// TwinCAT 3 PLC project PLC1
// ProgramVersion: 3.1.4023.0
// libraries:
//   Tc2_ModbusRTU, * (Beckhoff Automation GmbH)
//   Tc2_Standard, * (Beckhoff Automation GmbH)
//   Tc2_System, * (Beckhoff Automation GmbH)
//   Tc2_Utilities, * (Beckhoff Automation GmbH)
//   Tc3_Module, * (Beckhoff Automation GmbH)
// project tree:
//   / PlcTask.TcTTO
//   POUs/ FB_ModbusMaster.TcPOU, FB_ModbusSlave.TcPOU, FB_PM2200.TcPOU, FB_TDS3000.TcPOU, I_ModbusSlave.TcIO, MAIN.TcPOU
// real-time tasks:
//   TASK PlcTask: cycle T#50us, priority 20, ADS port 350
// I/O:
//   DEVICE Device 1 (COM Port)
//   DEVICE Device 2 (EtherCAT), AmsNetId 192.168.56.1.3.1
//     Term 1 (EK1100) [EK1100 EtherCAT Coupler (2A E-Bus)]
//       Term 2 (EL6022) [EL6022 Interface 2Ch. (RS422/485)]
// variable links:
//   PLC1/PLC1 Instance <-> Device 1 (COM Port)
//     PlcTask Inputs/MAIN.fbModbusMaster.fbModbusMaster.InData/D <-> Inputs/Data1
//     PlcTask Inputs/MAIN.fbModbusMaster.fbModbusMaster.InData/D @bit {8..504 step 8} <-> Inputs/Data{2..64}  (63 links)
//     PlcTask Inputs/MAIN.fbModbusMaster.fbModbusMaster.InData/SerStatus <-> Inputs/Status
//     PlcTask Outputs/MAIN.fbModbusMaster.fbModbusMaster.OutData/D <-> Outputs/Data1
//     PlcTask Outputs/MAIN.fbModbusMaster.fbModbusMaster.OutData/D @bit {8..504 step 8} <-> Outputs/Data{2..64}  (63 links)
//     PlcTask Outputs/MAIN.fbModbusMaster.fbModbusMaster.OutData/SerCtrl <-> Outputs/Ctrl

CONFIGURATION PLC1
    RESOURCE PLC ON TwinCAT3
        TASK PlcTask(INTERVAL := T#50us, PRIORITY := 20);
        PROGRAM MAIN WITH PlcTask : MAIN;
    END_RESOURCE
END_CONFIGURATION

// ---- POUs/I_ModbusSlave.TcIO
INTERFACE I_ModbusSlave

PROPERTY Address : POINTER TO WORD
GET
END_GET
END_PROPERTY

METHOD Convert : BOOL
VAR_INPUT
	iRegionNo	:	INT;
	pReadData	:	POINTER TO BYTE;
END_VAR
END_METHOD

METHOD FirstCycle : BOOL
VAR_INPUT
END_VAR
END_METHOD

PROPERTY Name : STRING
GET
END_GET
SET
END_SET
END_PROPERTY

PROPERTY NumAddRegion : UINT
GET
END_GET
END_PROPERTY

PROPERTY UnitID : BYTE
GET
END_GET
SET
END_SET
END_PROPERTY

END_INTERFACE

// ---- POUs/MAIN.TcPOU
PROGRAM MAIN
VAR
	fbModbusMaster 	:		FB_ModbusMaster;
	fbModbusSlave	:		FB_PM2200;
	fbModbusTemp	: 		FB_TDS3000;
	istep			:		UINT;
	bStart			:		BOOL;
	
	arrData			:		ARRAY [0..255] OF BYTE;
END_VAR

CASE istep OF
	0: //Trigger
		IF bStart THEN
			bStart := FALSE;
			istep := 10;
		END_IF
		
	10: //Init
		fbModbusSlave.UnitID := 1;
		fbModbusSlave.FirstCycle();
		fbModbusTemp.UnitID := 2;
		fbModbusTemp.FirstCycle();
		
		fbModbusMaster.FirstCycle();
		fbModbusMaster.Init();
		fbModbusMaster.RegisterSlave(fbModbusSlave);
		fbModbusMaster.RegisterSlave(fbModbusTemp);
		fbModbusMaster.Timeout := 1000;
		istep := 20;
		
	20: //Running
		IF fbModbusMaster.Run() THEN
			istep := 30;
		END_IF
		
	30: //Stopped
		
END_CASE

fbModbusMaster();

END_PROGRAM

// ---- POUs/FB_ModbusMaster.TcPOU
FUNCTION_BLOCK FB_ModbusMaster //IMPLEMENTS I_UniversalUnit
VAR
	sName			:		STRING;
	bInitialized	:		BOOL;
	iScantime		:		UINT;
	iTimeout		:		UINT;
	iErrorID		:		UDINT;
	
	bBusy			: 		BOOL;
	bError			:		BOOL;
	
	iStepInit		:		INT;
	iStepGeneral	: 		INT;
	iStepRunning	:		INT;
	bFirstCycle		:		BOOL;
	
	bRun			:		BOOL;
	bStop			: 		BOOL;
	
	fbModbusMaster	: 		ModbusRtuMaster_PcCOM;
	ipModbusSlave	:		ARRAY [1..247] OF I_ModbusSlave;
	iAmountSlave	: 		UINT;
	
	iLoopSlave		:		UINT	:= 1;
	iLoopAdr		:		UINT;
	iQuantity 		: 		POINTER TO WORD;
	iMBAddr 		: 		POINTER TO WORD;
    arrData			: 		ARRAY [0..255] OF BYTE;
	
END_VAR

IF bFirstCycle THEN
	bFirstCycle := FALSE;
END_IF
		
StateMachine();

bRun := FALSE;
bStop := FALSE;

bInitialized := iStepGeneral >= 20;

bError := fbModbusMaster.Error AND iStepGeneral = 30;
iErrorID := fbModbusMaster.ErrorId;
bBusy := fbModbusMaster.BUSY AND iStepGeneral = 30;

//	// error	
//		fbAxisError.Description := FUN_MergeStrings5(sMotorName, ' axis error number: ', UDINT_TO_STRING(iErrorID), '', '');
//		fbAxisError.Set(bError);

METHOD Abort : BOOL
END_METHOD

PROPERTY AnyError : BOOL
GET
AnyError 	:= bError;
END_GET
END_PROPERTY

PROPERTY Busy : BOOL
GET
Busy := bBusy;
END_GET
END_PROPERTY

PROPERTY ErrorID : UDINT
GET
ErrorID := iErrorID;
END_GET
END_PROPERTY

METHOD FirstCycle : BOOL
VAR_INPUT
//	ipAlarmController	: I_AlarmController;
//	ipHMIController	: I_HMIController;
END_VAR
END_METHOD

METHOD Init : BOOL
IF iStepGeneral = 0 THEN
	iStepGeneral := 10;
END_IF

//Method output
	Init := (iStepGeneral >= 20);
END_METHOD

PROPERTY Initialized : BOOL
GET
Initialized := bInitialized;
END_GET
END_PROPERTY

PROPERTY Name : STRING
GET
Name := sName;
END_GET
SET
sName := Name;
END_SET
END_PROPERTY

PROPERTY ReadData : ARRAY [0..255] OF BYTE
GET
ReadData := arrData;
END_GET
END_PROPERTY

PROPERTY ReadDataSize : uint
GET
ReadDataSize := INT_TO_UINT(SIZEOF(arrData));
END_GET
END_PROPERTY

METHOD RegisterSlave : BOOL
VAR_INPUT
	ModbusSlave		:		I_ModbusSlave;
END_VAR
VAR
	iLoop	:	UINT;
	bExists	:	BOOL;
END_VAR
FOR iLoop := 1 TO iAmountSlave DO
	IF ipModbusSlave[iLoop] = ModbusSlave THEN
		bExists := TRUE;
		iLoop := iAmountSlave;
	END_IF
END_FOR 
IF NOT bExists THEN
	iAmountSlave := iAmountSlave + 1;
	ipModbusSlave[iAmountSlave] := ModbusSlave;
END_IF
END_METHOD

METHOD Reset : BOOL
bError := FALSE;
iErrorID := 0;
bError := FALSE;
iStepInit		:= 0;
iStepGeneral	:= 0;
iStepRunning	:= 0;

iLoopSlave		:= 1;
iLoopAdr		:= 0;

fbModbusMaster.Execute := FALSE;

Reset := TRUE;
END_METHOD

METHOD Run : BOOL
IF (iStepGeneral = 20) THEN
	iStepGeneral := 30;
END_IF

bRun := TRUE;
Run := (iStepGeneral >= 30) AND (iStepGeneral < 200);
END_METHOD

PROPERTY ScanTime : UINT
GET
ScanTime := iScantime;
END_GET
SET
iScantime := ScanTime;
END_SET
END_PROPERTY

METHOD StateInit : BOOL (*Unit is performing initialization*)
IF NOT bError THEN
	iStepGeneral := 20;
END_IF
END_METHOD

METHOD StateMachine : BOOL (*State machine of unit*)
//State machine						   
	CASE iStepGeneral OF
		0:  //Uninitialized
			StateUninitialized();
	
		10: //Initializing
			StateInit();
	
		20: //Ready
			StateReady();
		
		30: //Running
			StateRunning();
						
		200: //stop
			StateStopping();
			
		210: //stop done
			StateStoppingDone();
	END_CASE
END_METHOD

METHOD StateReady : BOOL (* Unit is initialized*)
END_METHOD

METHOD StateRunning : BOOL (* Unit is uninitialized*)
VAR 
END_VAR
CASE iStepRunning OF
	0: // Trigger
		IF iAmountSlave > 0 THEN
			iStepRunning := 10;
		ELSE
			iStepRunning := 50;
		END_IF
		
	10: // Set parameters
		IF iLoopSlave <= iAmountSlave THEN
			IF  iLoopAdr <= ipModbusSlave[iLoopSlave].NumAddRegion - 1 THEN
				iQuantity := (ipModbusSlave[iLoopSlave].Address + (iLoopAdr*2+1)*SIZEOF(WORD));
				iMBAddr := (ipModbusSlave[iLoopSlave].Address + (iLoopAdr*2)*SIZEOF(WORD));
				
				fbModbusMaster.UnitID 	:=		ipModbusSlave[iLoopSlave].UnitID;
				fbModbusMaster.Quantity	:=		iQuantity^;
				fbModbusMaster.MBAddr	:=		iMBAddr^;
				fbModbusMaster.cbLength	:= 		SIZEOF(arrData);
				fbModbusMaster.pMemoryAddr	:= 	ADR(arrData);
				fbModbusMaster.Timeout	:= 		UINT_TO_TIME(iTimeout);
				
				iLoopAdr := iLoopAdr + 1;
			ELSE
				iLoopAdr := 0;
				iLoopSlave := iLoopSlave + 1;
			END_IF
		ELSE
			iLoopSlave := 1;
		END_IF
		iStepRunning := 20;
		
	20: // Send request
		IF NOT fbModbusMaster.BUSY THEN
			iStepRunning := 30;
		END_IF
	
	30: // Wait ack request
		IF fbModbusMaster.BUSY THEN
			iStepRunning := 40;
		END_IF
		
	40: // Wait respond
		IF NOT fbModbusMaster.BUSY THEN
			iStepRunning := 50;
		END_IF
		
	50: // Convert raw data
		ipModbusSlave[iLoopSlave].Convert(iLoopAdr, ADR(arrData));

	60: // Return, done
		iStepRunning := 0;
		
END_CASE

IF (iStepRunning >= 20) AND (iStepRunning <= 40) THEN
	fbModbusMaster.ReadRegs();
END_IF
fbModbusMaster.Execute := iStepRunning >= 20 AND iStepRunning <= 30;


//bTest S= iStepRunning > 
//tonTest(IN :=
END_METHOD

METHOD StateStopping : BOOL (* Unit is uninitialized*)
iStepGeneral	:= 0;
iStepRunning	:= 210;

iLoopSlave		:= 1;
iLoopAdr		:= 0;

fbModbusMaster.Execute := FALSE;
END_METHOD

METHOD StateStoppingDone : BOOL (* Unit is uninitialized*)
IF NOT bStop THEN
	iStepGeneral := 20;
END_IF
END_METHOD

METHOD StateUninitialized : BOOL (* Unit is uninitialized*)
END_METHOD

METHOD Stop : BOOL
IF iStepGeneral >= 30 AND iStepGeneral < 200 THEN
	iStepGeneral := 200;
END_IF
bStop := TRUE;

Stop := (iStepGeneral = 210);
END_METHOD

PROPERTY Timeout : UINT
GET
Timeout := iTimeout;
END_GET
SET
iTimeout := Timeout;
END_SET
END_PROPERTY

END_FUNCTION_BLOCK

// ---- POUs/FB_PM2200.TcPOU
FUNCTION_BLOCK FB_PM2200 EXTENDS FB_ModbusSlave
VAR
	arrAccPower	:	ARRAY [0..41] OF WORD;
	arrQuaPower		:	ARRAY [0..17] OF WORD;
	arrCommon		:	ARRAY [0..111] OF WORD;
END_VAR

PROPERTY AccPower : ARRAY [0..41] OF WORD
GET
AccPower := arrAccPower;
END_GET
END_PROPERTY

PROPERTY Common : ARRAY [0..111] OF WORD
GET
Common := arrCommon;
END_GET
END_PROPERTY

METHOD Convert : BOOL
VAR_INPUT
	iRegionNo	:	INT;
	pReadData	:	POINTER TO BYTE;
END_VAR
VAR
	pTempData	: 	POINTER TO BYTE;
	iTempData	: 	BYTE;
	iLoop		: 	INT;
	bHiByte		:	BOOL := TRUE;
END_VAR
CASE iRegionNo OF
	0: 
		FOR iLoop := 0 TO SIZEOF(arrAccPower)*2 DO
			pTempData := (pReadData + iLoop);
			iTempData := pTempData^;
			
			IF bHiByte THEN
				arrAccPower[iLoop/2] := SHL(BYTE_TO_WORD(iTempData), 8);
			ELSE 
				arrAccPower[iLoop/2] := arrAccPower[iLoop/2] + BYTE_TO_WORD(iTempData);
				IF bSwap THEN
					arrAccPower[iLoop/2] := ROL(arrAccPower[iLoop/2], 8);
				END_IF
			END_IF
			bHiByte := NOT bHiByte;
		END_FOR
		
	1: 
		FOR iLoop := 0 TO SIZEOF(arrQuaPower)*2 DO
			pTempData := (pReadData + iLoop);
			iTempData := pTempData^;
			
			IF bHiByte THEN
				arrQuaPower[iLoop/2] := SHL(BYTE_TO_WORD(iTempData), 8);
			ELSE 
				arrQuaPower[iLoop/2] := arrQuaPower[iLoop/2] + BYTE_TO_WORD(iTempData);
				IF bSwap THEN
					arrQuaPower[iLoop/2] := ROL(arrQuaPower[iLoop/2], 8);
				END_IF
			END_IF
			bHiByte := NOT bHiByte;
		END_FOR

	2: 
		FOR iLoop := 0 TO SIZEOF(arrCommon)*2 DO
			pTempData := (pReadData + iLoop);
			iTempData := pTempData^;
			
			IF bHiByte THEN
				arrCommon[iLoop/2] := SHL(BYTE_TO_WORD(iTempData), 8);
			ELSE 
				arrCommon[iLoop/2] := arrCommon[iLoop/2] + BYTE_TO_WORD(iTempData);
				IF bSwap THEN
					arrCommon[iLoop/2] := ROL(arrCommon[iLoop/2], 8);
				END_IF
			END_IF
			bHiByte := NOT bHiByte;
		END_FOR

END_CASE
END_METHOD

METHOD FirstCycle : BOOL
VAR_INPUT
END_VAR
arrAddress[0][0] := 2999;			// Current
arrAddress[0][1] := 12;

arrAddress[1][0] := 3019;			// Voltage
arrAddress[1][1] := 14;		
		
arrAddress[2][0] := 3053;
arrAddress[2][1] := 16;				// Power
arrAddress[3][0] := 3069;
arrAddress[3][1] := 8;				

arrAddress[4][0] := 3077;			// Power factor
arrAddress[4][1] := 16;		
		
arrAddress[5][0] := 3109;			// Frequency
arrAddress[6][1] := 2;				

iNumAddRegion := 6;
END_METHOD

PROPERTY QuaPower : ARRAY [0..17] OF WORD
GET
QuaPower := arrQuaPower;
END_GET
END_PROPERTY

END_FUNCTION_BLOCK

// ---- POUs/FB_ModbusSlave.TcPOU
FUNCTION_BLOCK FB_ModbusSlave IMPLEMENTS I_ModbusSlave
VAR
	iUnitID			: 		BYTE;
	arrAddress		:		ARRAY [0..20] OF ARRAY [0..1] OF WORD;
	iNumAddRegion	:		UINT;
	bSwap			:		BOOL;
	
	sName			:		STRING;

END_VAR

PROPERTY Address : POINTER TO WORD
GET
Address := ADR(arrAddress);
END_GET
END_PROPERTY

METHOD Convert : BOOL
VAR_INPUT
	iRegionNo	:	INT;
	pReadData	:	POINTER TO BYTE;
END_VAR
END_METHOD

METHOD FirstCycle : BOOL
VAR_INPUT
END_VAR
END_METHOD

PROPERTY Name : STRING
GET
Name := sName;
END_GET
SET
sName := Name;
END_SET
END_PROPERTY

PROPERTY NumAddRegion : UINT
GET
NumAddRegion := iNumAddRegion;
END_GET
END_PROPERTY

PROPERTY UnitID : BYTE
GET
UnitID := iUnitID;
END_GET
SET
iUnitID := UnitID;
END_SET
END_PROPERTY

END_FUNCTION_BLOCK

// ---- POUs/FB_TDS3000.TcPOU
FUNCTION_BLOCK FB_TDS3000 EXTENDS FB_ModbusSlave
VAR
	arrConditionData	:	ARRAY [0..63] OF WORD;
	arrUp_LoLimit		:	ARRAY [0..63] OF WORD;
	arrUpUp_UpLimit		:	ARRAY [0..63] OF WORD;
END_VAR

PROPERTY ConditionData : ARRAY [0..63] OF WORD
GET
ConditionData := arrConditionData;
END_GET
END_PROPERTY

METHOD Convert : BOOL
VAR_INPUT
	iRegionNo	:	INT;
	pReadData	:	POINTER TO BYTE;
END_VAR
VAR
	pTempData	: 	POINTER TO BYTE;
	iTempData	: 	BYTE;
	iLoop		: 	INT;
	bHiByte		:	BOOL := TRUE;
END_VAR
CASE iRegionNo OF
	0: 
		FOR iLoop := 0 TO SIZEOF(arrAddress[0][1])*2 DO
			pTempData := (pReadData + iLoop);
			iTempData := pTempData^;
			
			IF bHiByte THEN
				arrConditionData[iLoop/2] := SHL(BYTE_TO_WORD(iTempData), 8);
			ELSE 
				arrConditionData[iLoop/2] := arrConditionData[iLoop/2] + BYTE_TO_WORD(iTempData);
				IF bSwap THEN
					arrConditionData[iLoop/2] := ROL(arrConditionData[iLoop/2], 8);
				END_IF
			END_IF
			bHiByte := NOT bHiByte;
		END_FOR
		
	1:
		FOR iLoop := 17 TO (SIZEOF(arrAddress[1][1])*2 + 17) DO
			pTempData := (pReadData + iLoop);
			iTempData := pTempData^;
			
			IF bHiByte THEN
				arrConditionData[iLoop/2] := SHL(BYTE_TO_WORD(iTempData), 8);
			ELSE 
				arrConditionData[iLoop/2] := arrConditionData[iLoop/2] + BYTE_TO_WORD(iTempData);
				IF bSwap THEN
					arrConditionData[iLoop/2] := ROL(arrConditionData[iLoop/2], 8);
				END_IF
			END_IF
			bHiByte := NOT bHiByte;
		END_FOR
		
	2: 
		FOR iLoop := 0 TO SIZEOF(arrAddress[2][1])*2 DO
			pTempData := (pReadData + iLoop);
			iTempData := pTempData^;
			
			IF bHiByte THEN
				arrUp_LoLimit[iLoop/2] := SHL(BYTE_TO_WORD(iTempData), 8);
			ELSE 
				arrUp_LoLimit[iLoop/2] := arrUp_LoLimit[iLoop/2] + BYTE_TO_WORD(iTempData);
				IF bSwap THEN
					arrUp_LoLimit[iLoop/2] := ROL(arrUp_LoLimit[iLoop/2], 8);
				END_IF
			END_IF
			bHiByte := NOT bHiByte;
		END_FOR
		
	3: 
		FOR iLoop := 17 TO SIZEOF(arrAddress[3][1])*2 + 17 DO
			pTempData := (pReadData + iLoop);
			iTempData := pTempData^;
			
			IF bHiByte THEN
				arrUp_LoLimit[iLoop/2] := SHL(BYTE_TO_WORD(iTempData), 8);
			ELSE 
				arrUp_LoLimit[iLoop/2] := arrUp_LoLimit[iLoop/2] + BYTE_TO_WORD(iTempData);
				IF bSwap THEN
					arrUp_LoLimit[iLoop/2] := ROL(arrUp_LoLimit[iLoop/2], 8);
				END_IF
			END_IF
			bHiByte := NOT bHiByte;
		END_FOR

	4: 
		FOR iLoop := 0 TO SIZEOF(arrAddress[4][1])*2 DO
			pTempData := (pReadData + iLoop);
			iTempData := pTempData^;
			
			IF bHiByte THEN
				arrUpUp_UpLimit[iLoop/2] := SHL(BYTE_TO_WORD(iTempData), 8);
			ELSE 
				arrUpUp_UpLimit[iLoop/2] := arrUpUp_UpLimit[iLoop/2] + BYTE_TO_WORD(iTempData);
				IF bSwap THEN
					arrUpUp_UpLimit[iLoop/2] := ROL(arrUpUp_UpLimit[iLoop/2], 8);
				END_IF
			END_IF
			bHiByte := NOT bHiByte;
		END_FOR

	5: 
		FOR iLoop := 17 TO SIZEOF(arrAddress[5][1])*2 + 17 DO
			pTempData := (pReadData + iLoop);
			iTempData := pTempData^;
			
			IF bHiByte THEN
				arrUpUp_UpLimit[iLoop/2] := SHL(BYTE_TO_WORD(iTempData), 8);
			ELSE 
				arrUpUp_UpLimit[iLoop/2] := arrUpUp_UpLimit[iLoop/2] + BYTE_TO_WORD(iTempData);
				IF bSwap THEN
					arrUpUp_UpLimit[iLoop/2] := ROL(arrUpUp_UpLimit[iLoop/2], 8);
				END_IF
			END_IF
			bHiByte := NOT bHiByte;
		END_FOR

END_CASE
END_METHOD

METHOD FirstCycle : BOOL
VAR_INPUT
END_VAR
arrAddress[0][0] := 16#0000;
arrAddress[0][1] := 17;
arrAddress[1][0] := 16#0017;
arrAddress[1][1] := 15;

arrAddress[2][0] := 16#0100;
arrAddress[2][1] := 17;
arrAddress[3][0] := 16#0117;
arrAddress[3][1] := 15;

arrAddress[4][0] := 16#0200;
arrAddress[4][1] := 17;
arrAddress[5][0] := 16#0217;
arrAddress[5][1] := 15;

iNumAddRegion := 6;

bSwap := TRUE;
END_METHOD

PROPERTY Up_LoLimit : ARRAY [0..63] OF WORD
GET
Up_LoLimit := arrUp_LoLimit;
END_GET
END_PROPERTY

PROPERTY UpUp_UpLimit : ARRAY [0..63] OF WORD
GET
UpUp_UpLimit := arrUpUp_UpLimit;
END_GET
END_PROPERTY

END_FUNCTION_BLOCK
